(* IEC 61131-3 sources: Word/plc-course/06-edges-and-one-shots/labs/solutions, 3 files *)

(* ---- 06-1-toggle-lamp.st ---- *)
(* Lab 06-1: One-button floodlight toggle (push-on / push-off).
   Module 06 (Edge detection and one-shots). REFERENCE SOLUTION - try the lab yourself first. *)

PROGRAM ToggleLamp
  VAR (* I/O - addresses follow the OpenPLC convention *)
    LightPB      AT %IX0.0 : BOOL;  (* Floodlight push-button, NO: TRUE while pressed *)
    LightsEnable AT %IX0.1 : BOOL;  (* Gatehouse key switch: TRUE = bay lighting enabled *)
    Floodlight   AT %QX0.0 : BOOL;  (* Floodlight contactor coil *)
  END_VAR
  VAR (* internal *)
    PressEdge : R_TRIG;             (* one-shot: TRUE for one scan when LightPB is pressed *)
  END_VAR

  (* 1. Detect the press. The edge detector is called on EVERY scan and never
        inside an IF, so its memory always follows the button, even while the
        lighting is disabled. A press that began while disabled has already
        been "used up" by the time the key switch comes back on. *)
  PressEdge(CLK := LightPB);

  (* 2. Act on the one-scan pulse, never on the level of the button.
        Holding the button keeps PressEdge.Q FALSE after the first scan,
        so the lamp cannot flicker. The disable wins over everything. *)
  IF NOT LightsEnable THEN
    Floodlight := FALSE;
  ELSIF PressEdge.Q THEN
    Floodlight := NOT Floodlight;
  END_IF;
END_PROGRAM

CONFIGURATION Config0
  RESOURCE Res0 ON PLC
    TASK MainTask(INTERVAL := T#10ms, PRIORITY := 0);
    PROGRAM Inst0 WITH MainTask : ToggleLamp;
  END_RESOURCE
END_CONFIGURATION

(* ---- 06-2-event-counter.st ---- *)
(* Lab 06-2: Carton and product-change counter (event counting and change-of-value).
   Module 06 (Edge detection and one-shots). REFERENCE SOLUTION - try the lab yourself first. *)

PROGRAM EventCounter
  VAR (* I/O - addresses follow the OpenPLC convention *)
    PartPE  AT %IX0.0 : BOOL;  (* Photo-eye: TRUE while a carton blocks the beam *)
    ResetPB AT %IX0.1 : BOOL;  (* Count reset push-button, NO: TRUE while pressed *)
  END_VAR
  VAR (* HMI values - part of the lab interface *)
    ProductSel : INT;          (* Product number selected by the operator on the HMI, 1..4 *)
    PartCount  : DINT;         (* Cartons counted since the last reset *)
    SelChanges : INT;          (* Changes of ProductSel since the last reset *)
  END_VAR
  VAR (* internal *)
    PartArrived : R_TRIG;      (* rising edge of the photo-eye = a carton has arrived *)
    SelPrev     : INT;         (* ProductSel as it was on the previous scan *)
    SelChanged  : BOOL;        (* TRUE for the one scan in which ProductSel changed *)
    Started     : BOOL;        (* FALSE at power-up, TRUE from the end of the first scan (not RETAIN) *)
    FirstScan   : BOOL;        (* TRUE during the first scan only *)
  END_VAR

  (* 1. Home-made first-scan flag. Started is not retentive, so it is FALSE
        after every power-up and FirstScan is TRUE for exactly one scan. *)
  FirstScan := NOT Started;
  Started := TRUE;

  (* 2. Edge and change detection run on EVERY scan, outside any IF, so their
        memories always follow the inputs - also while Reset is held. *)
  PartArrived(CLK := PartPE);

  SelChanged := ProductSel <> SelPrev;
  SelPrev := ProductSel;               (* remember for the next scan - always LAST *)

  (* 3. Whatever the inputs are at power-up is the starting point, not an event:
        a carton already blocking the beam has not just "arrived", and the
        selector's power-up position is not a change. *)
  IF FirstScan THEN
    SelChanged := FALSE;
  END_IF;

  (* 4. Counting. Reset is level-sensitive and has priority: while it is held
        the counts stay at zero and events are discarded. *)
  IF ResetPB THEN
    PartCount := 0;
    SelChanges := 0;
  ELSE
    IF PartArrived.Q AND NOT FirstScan THEN
      PartCount := PartCount + 1;
    END_IF;
    IF SelChanged THEN
      SelChanges := SelChanges + 1;
    END_IF;
  END_IF;
END_PROGRAM

CONFIGURATION Config0
  RESOURCE Res0 ON PLC
    TASK MainTask(INTERVAL := T#10ms, PRIORITY := 0);
    PROGRAM Inst0 WITH MainTask : EventCounter;
  END_RESOURCE
END_CONFIGURATION

(* ---- 06-3-duty-standby.st ---- *)
(* Lab 06-3: Duty-standby pump alternation.
   Module 06 (Edge detection and one-shots). REFERENCE SOLUTION - try the lab yourself first.
   Training exercise only: a real pump station also needs level alarms, run
   feedback, start delays and a design review (Modules 07, 14, 16). *)

PROGRAM DutyStandby
  VAR (* I/O - addresses follow the OpenPLC convention *)
    Demand     AT %IX0.0 : BOOL;  (* Pumping demand from the sump level control: TRUE = pump needed *)
    Pump1OK_NC AT %IX0.1 : BOOL;  (* Pump 1 healthy (overload relay + motor protection), NC: TRUE when healthy *)
    Pump2OK_NC AT %IX0.2 : BOOL;  (* Pump 2 healthy, NC: TRUE when healthy *)
    Pump1      AT %QX0.0 : BOOL;  (* Pump 1 contactor *)
    Pump2      AT %QX0.1 : BOOL;  (* Pump 2 contactor *)
  END_VAR
  VAR (* internal *)
    NewDemand : R_TRIG;           (* one-shot: a new demand has just started *)
    SelectP2  : BOOL;             (* FALSE = Pump 1 selected, TRUE = Pump 2 selected *)
    LastRanP1 : BOOL;             (* TRUE = Pump 1 ran last; FALSE = Pump 2 ran last, or none yet *)
  END_VAR

  (* 1. Alternation - only on the EDGE of a new demand. Choosing on the level
        would swap pumps on every scan while the demand lasts.
        At power-up SelectP2 is FALSE, so Pump 1 is selected even if the edge
        detector does not fire on the first scan (not every platform's does). *)
  NewDemand(CLK := Demand);
  IF NewDemand.Q THEN
    SelectP2 := LastRanP1;        (* the pump that did NOT run last time *)
  END_IF;

  (* 2. Fault handling - checked on every scan. If the selected pump is not
        healthy and the other one is, move the selection to the other pump.
        Nothing moves the selection back when the fault clears, so a pump
        that has taken over keeps running until the demand ends (no bumping). *)
  IF SelectP2 AND NOT Pump2OK_NC AND Pump1OK_NC THEN
    SelectP2 := FALSE;
  ELSIF NOT SelectP2 AND NOT Pump1OK_NC AND Pump2OK_NC THEN
    SelectP2 := TRUE;
  END_IF;

  (* 3. Outputs. The selection is a single BOOL, so both pumps can never be
        commanded at the same time. A faulted pump is never commanded. *)
  Pump1 := Demand AND NOT SelectP2 AND Pump1OK_NC;
  Pump2 := Demand AND SelectP2 AND Pump2OK_NC;

  (* 4. Remember which pump actually ran, for the next alternation. *)
  IF Pump1 THEN
    LastRanP1 := TRUE;
  ELSIF Pump2 THEN
    LastRanP1 := FALSE;
  END_IF;
END_PROGRAM

CONFIGURATION Config0
  RESOURCE Res0 ON PLC
    TASK MainTask(INTERVAL := T#10ms, PRIORITY := 0);
    PROGRAM Inst0 WITH MainTask : DutyStandby;
  END_RESOURCE
END_CONFIGURATION
